% RSLogix 500 project LEGACY DRYER WITH LONOX AND SHUTDOWN DELAY.RSS, saved by version 11.00.00.00 %
PROJECT "ML1200"    % processor: MicroLogix 1200; MAIN_PROG %

PROGRAM FILES
  LAD 2 "MAIN_PROG"  15 rungs
  LAD 3 "DRYER CONT"  18 rungs
  LAD 4 "TEMPERATUR"  33 rungs
  LAD 5 "AIR PRES."  12 rungs
  LAD 6 "HUMIDITY"  14 rungs
  LAD 7 "RHL-TEMP"  2 rungs  % HEATING CONTROLS %
  LAD 8 "HEAT CONTR"  47 rungs
  LAD 9 "CLR FAULTS"  2 rungs
  LAD 10 "HOUR METER"  5 rungs
  LAD 11 "CONV CLEAN"  14 rungs

DATA FILES
  O0 OUTPUT  8 elements
  I1 INPUT  19 elements
  S2 STATUS  66 elements
  B3 BINARY  20 elements
  T4 TIMER  13 elements
  C5 COUNTER  1 elements
  R6 CONTROL  1 elements
  N7 INTEGER  77 elements
  F8 FLOAT  1 elements
  PD9 DRYER  3 elements

LADDER 2 "MAIN_PROG"
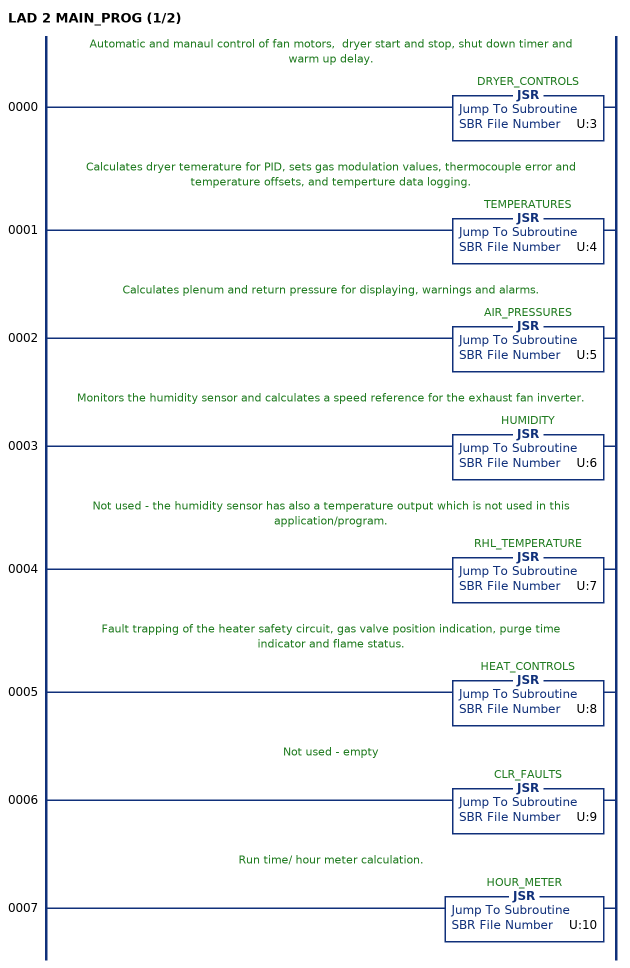
% Rung: 0 %
% Automatic and manaul control of fan motors,  dryer start and stop, shut down timer and warm up delay. %
SOR JSR U:3 EOR
%   U:3  DRYER_CONTROLS %
% Rung: 1 %
% Calculates dryer temerature for PID, sets gas modulation values, thermocouple error and temperature offsets, and temperture data logging. %
SOR JSR U:4 EOR
%   U:4  TEMPERATURES %
% Rung: 2 %
% Calculates plenum and return pressure for displaying, warnings and alarms. %
SOR JSR U:5 EOR
%   U:5  AIR_PRESSURES %
% Rung: 3 %
% Monitors the humidity sensor and calculates a speed reference for the exhaust fan inverter. %
SOR JSR U:6 EOR
%   U:6  HUMIDITY %
% Rung: 4 %
% Not used - the humidity sensor has also a temperature output which is not used in this application/program. %
SOR JSR U:7 EOR
%   U:7  RHL_TEMPERATURE %
% Rung: 5 %
% Fault trapping of the heater safety circuit, gas valve position indication, purge time indicator and flame status. %
SOR JSR U:8 EOR
%   U:8  HEAT_CONTROLS %
% Rung: 6 %
% Not used - empty %
SOR JSR U:9 EOR
%   U:9  CLR_FAULTS %
% Rung: 7 %
% Run time/ hour meter calculation. %
SOR JSR U:10 EOR
%   U:10  HOUR_METER %

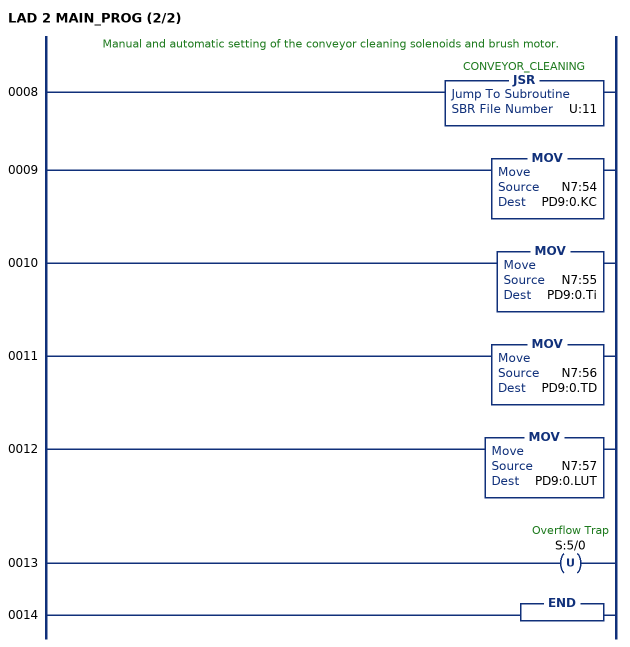
% Rung: 8 %
% Manual and automatic setting of the conveyor cleaning solenoids and brush motor. %
SOR JSR U:11 EOR
%   U:11  CONVEYOR_CLEANING %
% Rung: 9 %
SOR MOV N7:54 PD9:0.KC EOR
%   N7:54  KC %
% Rung: 10 %
SOR MOV N7:55 PD9:0.Ti EOR
%   N7:55  TI %
% Rung: 11 %
SOR MOV N7:56 PD9:0.TD EOR
%   N7:56  TD %
% Rung: 12 %
SOR MOV N7:57 PD9:0.LUT EOR
%   N7:57  LUT %
% Rung: 13 %
SOR OTU S:5/0 EOR
%   S:5/0  "Overflow Trap" %
% Rung: 14 %
SOR END EOR

LADDER 3 "DRYER CONT"
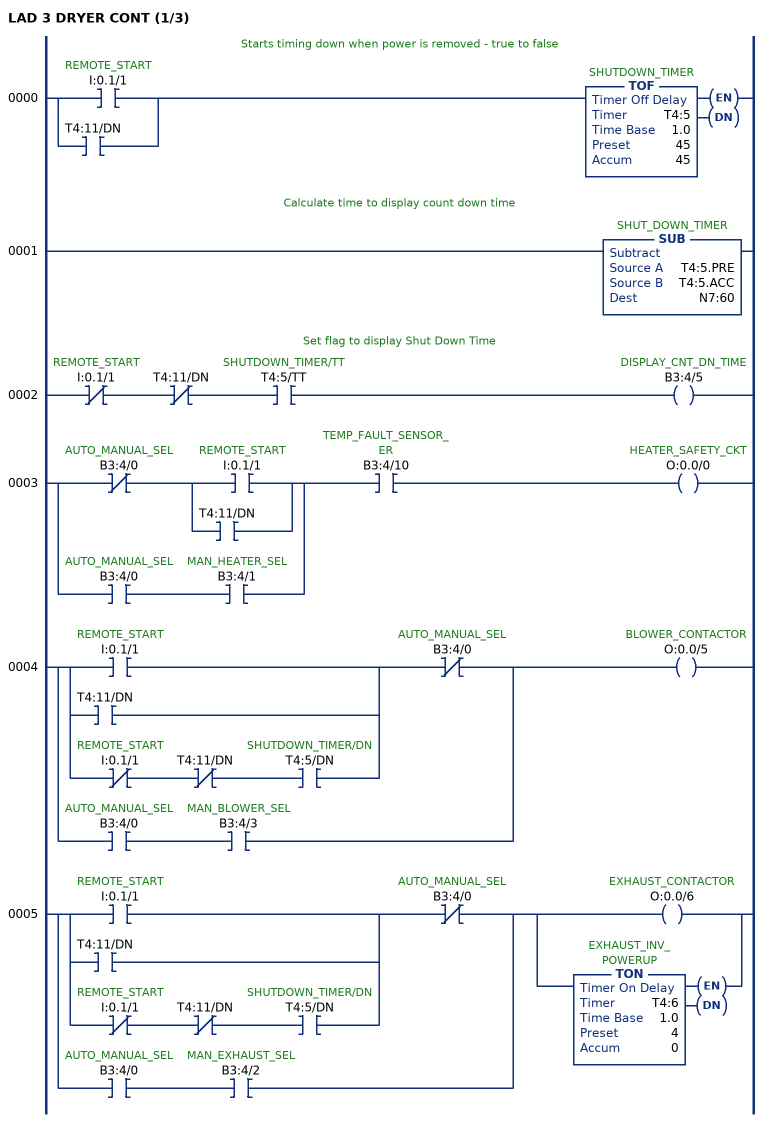
% Rung: 0 %
% Starts timing down when power is removed - true to false %
SOR BST XIC I:0.1/1 NXB XIC T4:11/DN BND TOF T4:5 1.0 45 45 EOR
%   I:0.1/1  REMOTE_START %
%   T4:5  SHUTDOWN_TIMER %
% Rung: 1 %
% Calculate time to display count down time %
SOR SUB T4:5.PRE T4:5.ACC N7:60 EOR
%   T4:5  SHUTDOWN_TIMER %
%   N7:60  SHUT_DOWN_TIMER %
% Rung: 2 %
% Set flag to display Shut Down Time %
SOR XIO I:0.1/1 XIO T4:11/DN XIC T4:5/TT OTE B3:4/5 EOR
%   I:0.1/1  REMOTE_START %
%   T4:5  SHUTDOWN_TIMER %
%   B3:4/5  DISPLAY_CNT_DN_TIME %
% Rung: 3 %
SOR BST XIO B3:4/0 BST XIC I:0.1/1 NXB XIC T4:11/DN BND NXB XIC B3:4/0 XIC B3:4/1 BND XIC B3:4/10 OTE O:0.0/0 EOR
%   B3:4/0  AUTO_MANUAL_SEL %
%   I:0.1/1  REMOTE_START %
%   B3:4/1  MAN_HEATER_SEL %
%   B3:4/10  TEMP_FAULT_SENSOR_ER %
%   O:0.0/0  HEATER_SAFETY_CKT %
% Rung: 4 %
SOR BST BST BST XIC I:0.1/1 NXB XIC T4:11/DN BND NXB XIO I:0.1/1 XIO T4:11/DN XIC T4:5/DN BND XIO B3:4/0 NXB XIC B3:4/0 XIC B3:4/3 BND OTE O:0.0/5 EOR
%   I:0.1/1  REMOTE_START %
%   T4:5  SHUTDOWN_TIMER %
%   B3:4/0  AUTO_MANUAL_SEL %
%   B3:4/3  MAN_BLOWER_SEL %
%   O:0.0/5  BLOWER_CONTACTOR %
% Rung: 5 %
SOR BST BST BST XIC I:0.1/1 NXB XIC T4:11/DN BND NXB XIO I:0.1/1 XIO T4:11/DN XIC T4:5/DN BND XIO B3:4/0 NXB XIC B3:4/0 XIC B3:4/2 BND BST OTE O:0.0/6 NXB TON T4:6 1.0 4 0 BND EOR
%   I:0.1/1  REMOTE_START %
%   T4:5  SHUTDOWN_TIMER %
%   B3:4/0  AUTO_MANUAL_SEL %
%   B3:4/2  MAN_EXHAUST_SEL %
%   O:0.0/6  EXHAUST_CONTACTOR %
%   T4:6  EXHAUST_INV_POWERUP %

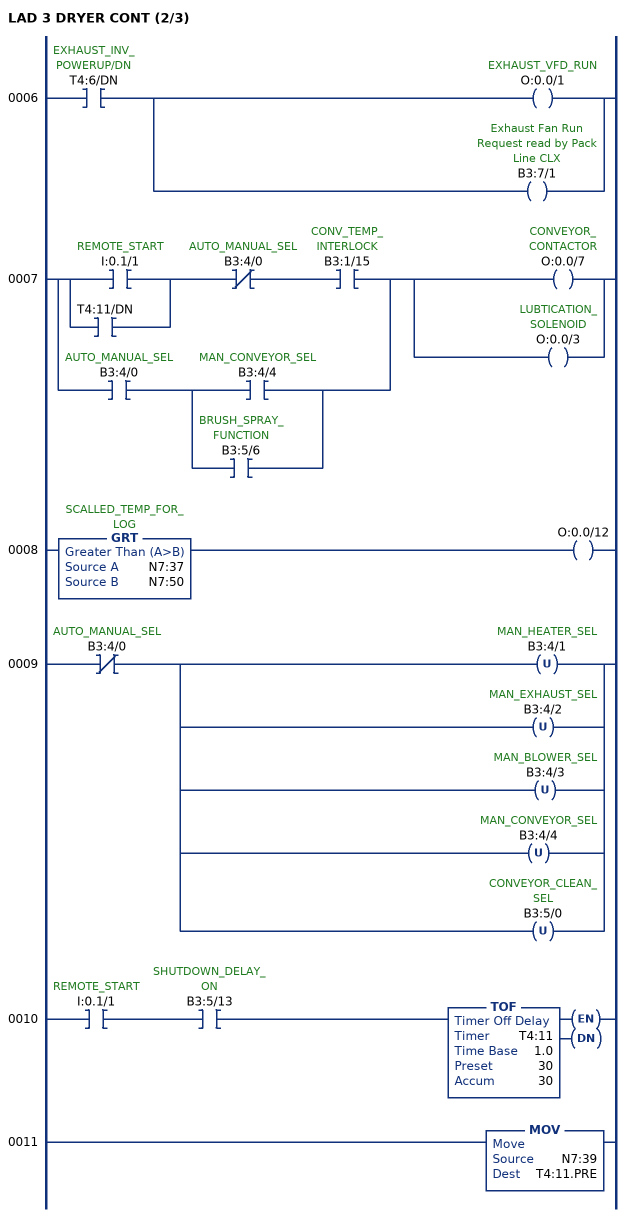
% Rung: 6 %
SOR XIC T4:6/DN BST OTE O:0.0/1 NXB OTE B3:7/1 BND EOR
%   T4:6  EXHAUST_INV_POWERUP %
%   O:0.0/1  EXHAUST_VFD_RUN %
%   B3:7/1  "Exhaust Fan Run Request read by Pack Line CLX" %
% Rung: 7 %
SOR BST BST XIC I:0.1/1 NXB XIC T4:11/DN BND XIO B3:4/0 XIC B3:1/15 NXB XIC B3:4/0 BST XIC B3:4/4 NXB XIC B3:5/6 BND BND BST OTE O:0.0/7 NXB OTE O:0.0/3 BND EOR
%   I:0.1/1  REMOTE_START %
%   B3:4/0  AUTO_MANUAL_SEL %
%   B3:1/15  CONV_TEMP_INTERLOCK %
%   B3:4/4  MAN_CONVEYOR_SEL %
%   B3:5/6  BRUSH_SPRAY_FUNCTION %
%   O:0.0/7  CONVEYOR_CONTACTOR %
%   O:0.0/3  LUBTICATION_SOLENOID %
% Rung: 8 %
SOR GRT N7:37 N7:50 OTE O:0.0/12 EOR
%   N7:37  SCALLED_TEMP_FOR_LOG %
% Rung: 9 %
SOR XIO B3:4/0 BST OTU B3:4/1 NXB BST OTU B3:4/2 NXB BST OTU B3:4/3 NXB BST OTU B3:4/4 NXB OTU B3:5/0 BND BND BND BND EOR
%   B3:4/0  AUTO_MANUAL_SEL %
%   B3:4/1  MAN_HEATER_SEL %
%   B3:4/2  MAN_EXHAUST_SEL %
%   B3:4/3  MAN_BLOWER_SEL %
%   B3:4/4  MAN_CONVEYOR_SEL %
%   B3:5/0  CONVEYOR_CLEAN_SEL %
% Rung: 10 %
SOR XIC I:0.1/1 XIC B3:5/13 TOF T4:11 1.0 30 30 EOR
%   I:0.1/1  REMOTE_START %
%   B3:5/13  SHUTDOWN_DELAY_ON %
% Rung: 11 %
SOR MOV N7:39 T4:11.PRE EOR

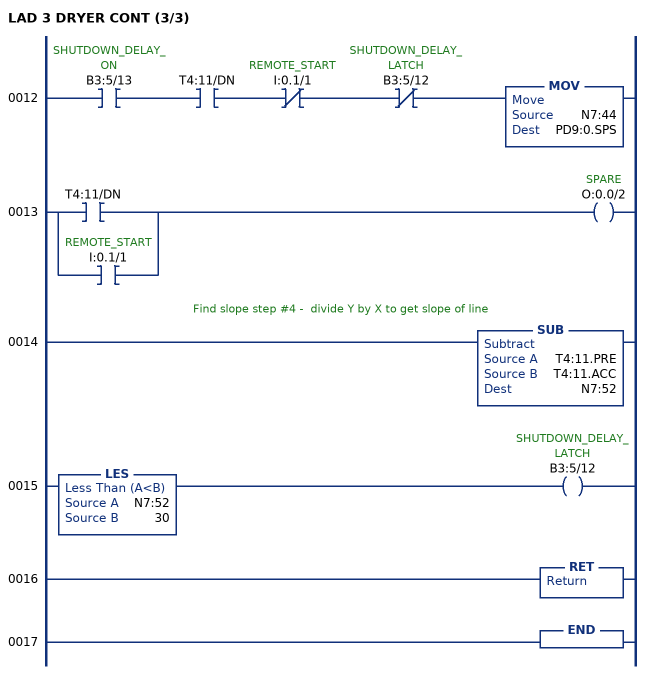
% Rung: 12 %
SOR XIC B3:5/13 XIC T4:11/DN XIO I:0.1/1 XIO B3:5/12 MOV N7:44 PD9:0.SPS EOR
%   B3:5/13  SHUTDOWN_DELAY_ON %
%   I:0.1/1  REMOTE_START %
%   B3:5/12  SHUTDOWN_DELAY_LATCH %
%   N7:44  TEMP_ON_SHUTDOWN_DLY %
% Rung: 13 %
SOR BST XIC T4:11/DN NXB XIC I:0.1/1 BND OTE O:0.0/2 EOR
%   I:0.1/1  REMOTE_START %
%   O:0.0/2  SPARE %
% Rung: 14 %
% Find slope step #4 -  divide Y by X to get slope of line %
SOR SUB T4:11.PRE T4:11.ACC N7:52 EOR
% Rung: 15 %
SOR LES N7:52 30 OTE B3:5/12 EOR
%   B3:5/12  SHUTDOWN_DELAY_LATCH %
% Rung: 16 %
SOR RET EOR
% Rung: 17 %
SOR END EOR

LADDER 4 "TEMPERATUR"
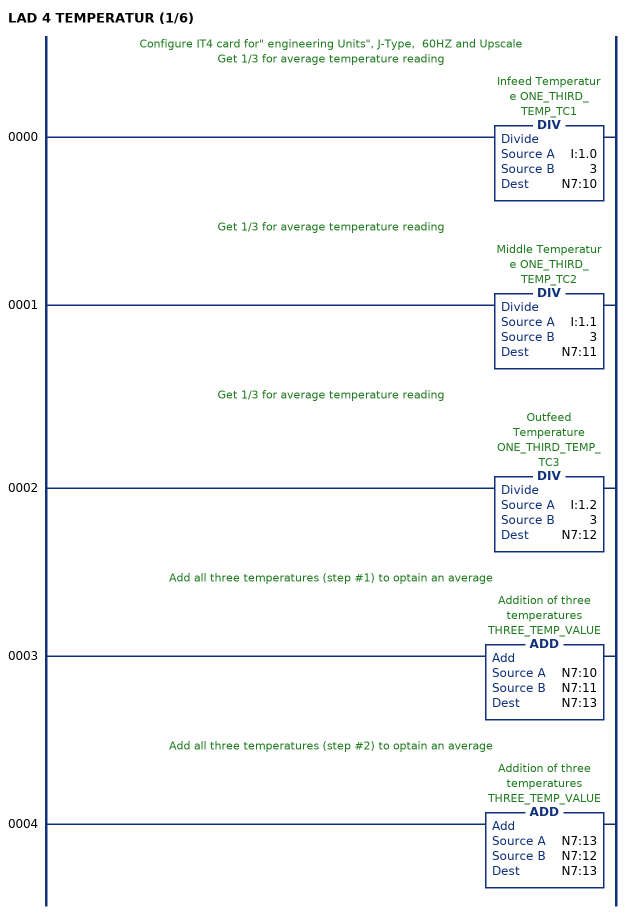
% Rung: 0 %
% Configure IT4 card for" engineering Units", J-Type,  60HZ and Upscale
% Get 1/3 for average temperature reading %
SOR DIV I:1.0 3 N7:10 EOR
%   I:1.0  INFEED_TEMP %
%   N7:10  ONE_THIRD_TEMP_TC1  "Infeed Temperature" %
% Rung: 1 %
% Get 1/3 for average temperature reading %
SOR DIV I:1.1 3 N7:11 EOR
%   I:1.1  MIDDLE_TEMP %
%   N7:11  ONE_THIRD_TEMP_TC2  "Middle Temperature" %
% Rung: 2 %
% Get 1/3 for average temperature reading %
SOR DIV I:1.2 3 N7:12 EOR
%   I:1.2  OUTFEED_TEMP %
%   N7:12  ONE_THIRD_TEMP_TC3  "Outfeed Temperature" %
% Rung: 3 %
% Add all three temperatures (step #1) to optain an average %
SOR ADD N7:10 N7:11 N7:13 EOR
%   N7:10  ONE_THIRD_TEMP_TC1  "Infeed Temperature" %
%   N7:11  ONE_THIRD_TEMP_TC2  "Middle Temperature" %
%   N7:13  THREE_TEMP_VALUE  "Addition of three temperatures" %
% Rung: 4 %
% Add all three temperatures (step #2) to optain an average %
SOR ADD N7:13 N7:12 N7:13 EOR
%   N7:13  THREE_TEMP_VALUE  "Addition of three temperatures" %
%   N7:12  ONE_THIRD_TEMP_TC3  "Outfeed Temperature" %

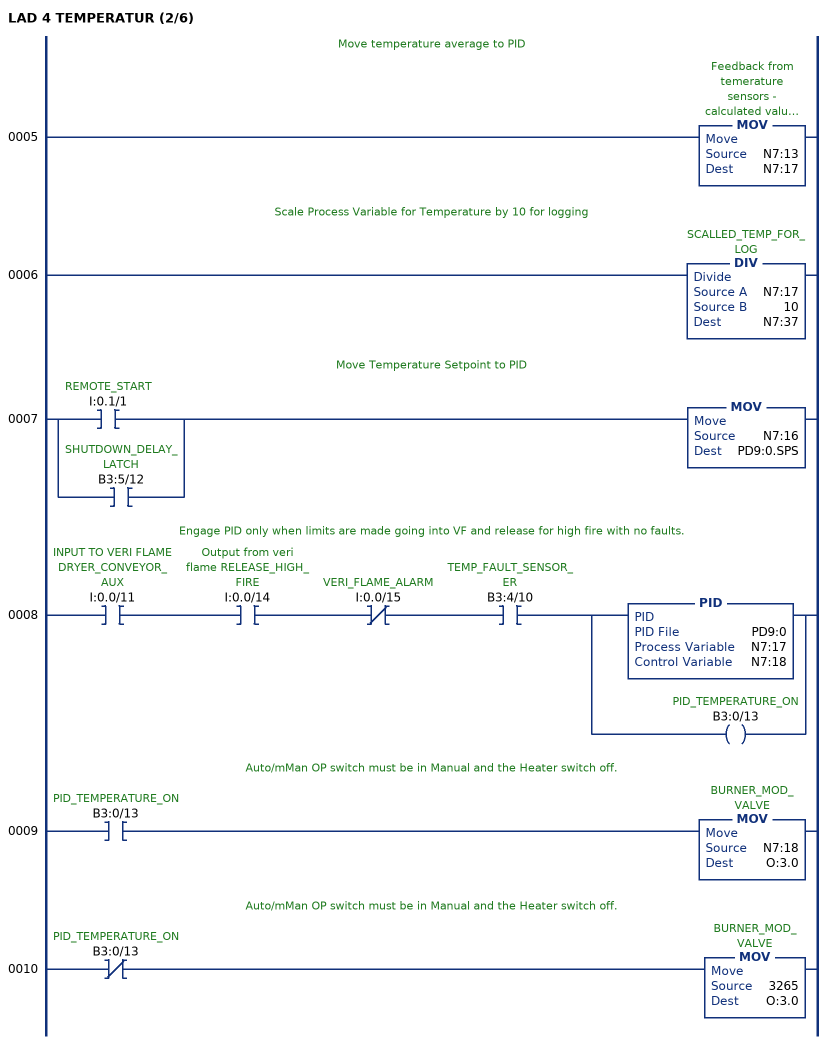
% Rung: 5 %
% Move temperature average to PID %
SOR MOV N7:13 N7:17 EOR
%   N7:13  THREE_TEMP_VALUE  "Addition of three temperatures" %
%   N7:17  PV_TEMP_PROCESS_VAR  "Feedback from temerature sensors - calculated value" %
% Rung: 6 %
% Scale Process Variable for Temperature by 10 for logging %
SOR DIV N7:17 10 N7:37 EOR
%   N7:17  PV_TEMP_PROCESS_VAR  "Feedback from temerature sensors - calculated value" %
%   N7:37  SCALLED_TEMP_FOR_LOG %
% Rung: 7 %
% Move Temperature Setpoint to PID %
SOR BST XIC I:0.1/1 NXB XIC B3:5/12 BND MOV N7:16 PD9:0.SPS EOR
%   I:0.1/1  REMOTE_START %
%   B3:5/12  SHUTDOWN_DELAY_LATCH %
%   N7:16  SPS_TEMP_SETPOINT  "Display Input Value - desired Temperature" %
% Rung: 8 %
% Engage PID only when limits are made going into VF and release for high fire with no faults. %
SOR XIC I:0.0/11 XIC I:0.0/14 XIO I:0.0/15 XIC B3:4/10 BST PID PD9:0 N7:17 N7:18 NXB OTE B3:0/13 BND EOR
%   I:0.0/11  DRYER_CONVEYOR_AUX  "INPUT TO VERI FLAME" %
%   I:0.0/14  RELEASE_HIGH_FIRE  "Output from veri flame" %
%   I:0.0/15  VERI_FLAME_ALARM %
%   B3:4/10  TEMP_FAULT_SENSOR_ER %
%   N7:17  PV_TEMP_PROCESS_VAR  "Feedback from temerature sensors - calculated value" %
%   N7:18  CV_TEMP_CONTROL_VAR  "Output value to output for output card" %
%   B3:0/13  PID_TEMPERATURE_ON %
% Rung: 9 %
% Auto/mMan OP switch must be in Manual and the Heater switch off. %
SOR XIC B3:0/13 MOV N7:18 O:3.0 EOR
%   B3:0/13  PID_TEMPERATURE_ON %
%   N7:18  CV_TEMP_CONTROL_VAR  "Output value to output for output card" %
%   O:3.0  BURNER_MOD_VALVE %
% Rung: 10 %
% Auto/mMan OP switch must be in Manual and the Heater switch off. %
SOR XIO B3:0/13 MOV 3265 O:3.0 EOR
%   B3:0/13  PID_TEMPERATURE_ON %
%   O:3.0  BURNER_MOD_VALVE %

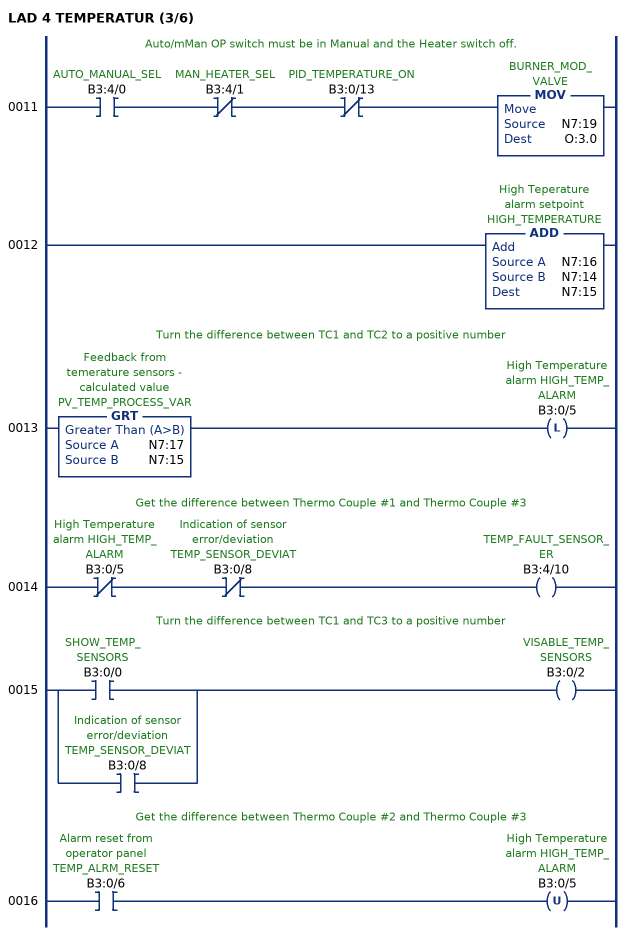
% Rung: 11 %
% Auto/mMan OP switch must be in Manual and the Heater switch off. %
SOR XIC B3:4/0 XIO B3:4/1 XIO B3:0/13 MOV N7:19 O:3.0 EOR
%   B3:4/0  AUTO_MANUAL_SEL %
%   B3:4/1  MAN_HEATER_SEL %
%   B3:0/13  PID_TEMPERATURE_ON %
%   N7:19  MANUAL_GAS_VALVE_POS  "To test burner butterfly in Manual" %
%   O:3.0  BURNER_MOD_VALVE %
% Rung: 12 %
SOR ADD N7:16 N7:14 N7:15 EOR
%   N7:16  SPS_TEMP_SETPOINT  "Display Input Value - desired Temperature" %
%   N7:14  HIGH_TEMP_OFFSET  "Value added to Temp Setpoint to set high temerature" %
%   N7:15  HIGH_TEMPERATURE  "High Teperature alarm setpoint" %
% Rung: 13 %
% Turn the difference between TC1 and TC2 to a positive number %
SOR GRT N7:17 N7:15 OTL B3:0/5 EOR
%   N7:17  PV_TEMP_PROCESS_VAR  "Feedback from temerature sensors - calculated value" %
%   N7:15  HIGH_TEMPERATURE  "High Teperature alarm setpoint" %
%   B3:0/5  HIGH_TEMP_ALARM  "High Temperature alarm" %
% Rung: 14 %
% Get the difference between Thermo Couple #1 and Thermo Couple #3 %
SOR XIO B3:0/5 XIO B3:0/8 OTE B3:4/10 EOR
%   B3:0/5  HIGH_TEMP_ALARM  "High Temperature alarm" %
%   B3:0/8  TEMP_SENSOR_DEVIAT  "Indication of sensor error/deviation" %
%   B3:4/10  TEMP_FAULT_SENSOR_ER %
% Rung: 15 %
% Turn the difference between TC1 and TC3 to a positive number %
SOR BST XIC B3:0/0 NXB XIC B3:0/8 BND OTE B3:0/2 EOR
%   B3:0/0  SHOW_TEMP_SENSORS %
%   B3:0/8  TEMP_SENSOR_DEVIAT  "Indication of sensor error/deviation" %
%   B3:0/2  VISABLE_TEMP_SENSORS %
% Rung: 16 %
% Get the difference between Thermo Couple #2 and Thermo Couple #3 %
SOR XIC B3:0/6 OTU B3:0/5 EOR
%   B3:0/6  TEMP_ALRM_RESET  "Alarm reset from operator panel" %
%   B3:0/5  HIGH_TEMP_ALARM  "High Temperature alarm" %

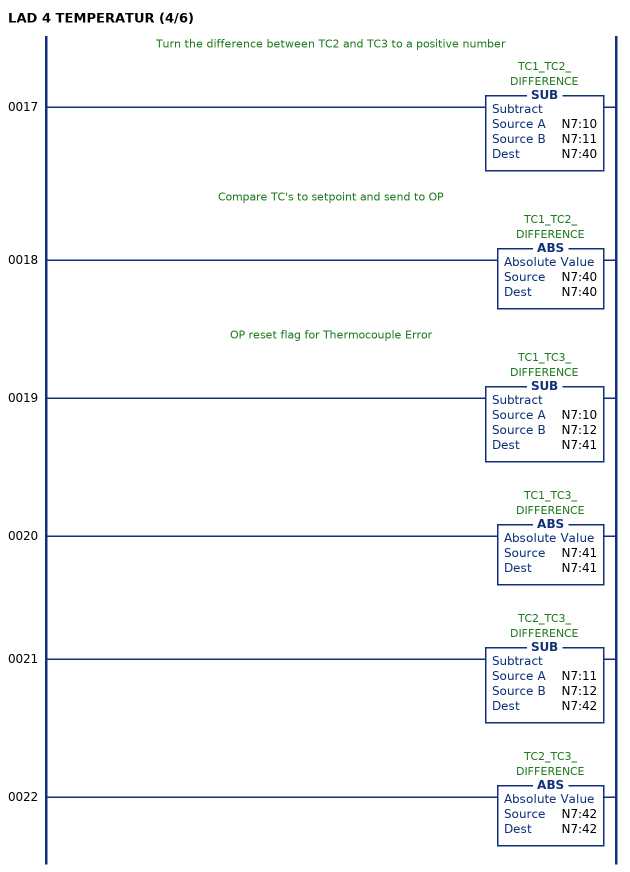
% Rung: 17 %
% Turn the difference between TC2 and TC3 to a positive number %
SOR SUB N7:10 N7:11 N7:40 EOR
%   N7:10  ONE_THIRD_TEMP_TC1  "Infeed Temperature" %
%   N7:11  ONE_THIRD_TEMP_TC2  "Middle Temperature" %
%   N7:40  TC1_TC2_DIFFERENCE %
% Rung: 18 %
% Compare TC's to setpoint and send to OP %
SOR ABS N7:40 N7:40 EOR
%   N7:40  TC1_TC2_DIFFERENCE %
% Rung: 19 %
% OP reset flag for Thermocouple Error %
SOR SUB N7:10 N7:12 N7:41 EOR
%   N7:10  ONE_THIRD_TEMP_TC1  "Infeed Temperature" %
%   N7:12  ONE_THIRD_TEMP_TC3  "Outfeed Temperature" %
%   N7:41  TC1_TC3_DIFFERENCE %
% Rung: 20 %
SOR ABS N7:41 N7:41 EOR
%   N7:41  TC1_TC3_DIFFERENCE %
% Rung: 21 %
SOR SUB N7:11 N7:12 N7:42 EOR
%   N7:11  ONE_THIRD_TEMP_TC2  "Middle Temperature" %
%   N7:12  ONE_THIRD_TEMP_TC3  "Outfeed Temperature" %
%   N7:42  TC2_TC3_DIFFERENCE %
% Rung: 22 %
SOR ABS N7:42 N7:42 EOR
%   N7:42  TC2_TC3_DIFFERENCE %

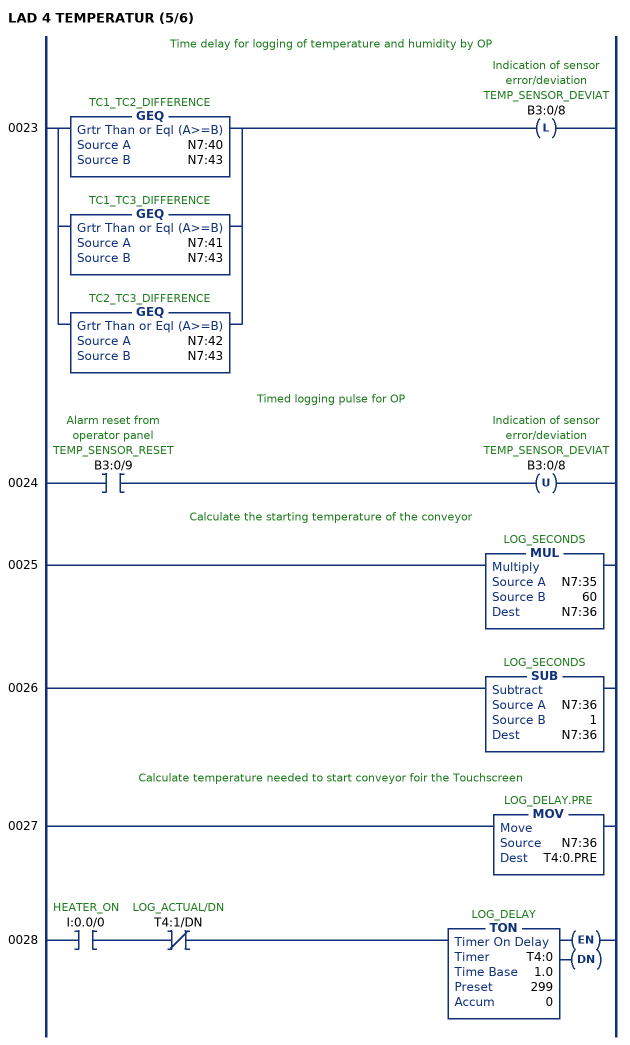
% Rung: 23 %
% Time delay for logging of temperature and humidity by OP %
SOR BST GEQ N7:40 N7:43 NXB BST GEQ N7:41 N7:43 NXB GEQ N7:42 N7:43 BND BND OTL B3:0/8 EOR
%   N7:40  TC1_TC2_DIFFERENCE %
%   N7:43  MAX_TEMP_SENSOR_DEV %
%   N7:41  TC1_TC3_DIFFERENCE %
%   N7:42  TC2_TC3_DIFFERENCE %
%   B3:0/8  TEMP_SENSOR_DEVIAT  "Indication of sensor error/deviation" %
% Rung: 24 %
% Timed logging pulse for OP %
SOR XIC B3:0/9 OTU B3:0/8 EOR
%   B3:0/9  TEMP_SENSOR_RESET  "Alarm reset from operator panel" %
%   B3:0/8  TEMP_SENSOR_DEVIAT  "Indication of sensor error/deviation" %
% Rung: 25 %
% Calculate the starting temperature of the conveyor %
SOR MUL N7:35 60 N7:36 EOR
%   N7:35  LOG_MINUTES %
%   N7:36  LOG_SECONDS %
% Rung: 26 %
SOR SUB N7:36 1 N7:36 EOR
%   N7:36  LOG_SECONDS %
% Rung: 27 %
% Calculate temperature needed to start conveyor foir the Touchscreen %
SOR MOV N7:36 T4:0.PRE EOR
%   N7:36  LOG_SECONDS %
%   T4:0  LOG_DELAY %
% Rung: 28 %
SOR XIC I:0.0/0 XIO T4:1/DN TON T4:0 1.0 299 0 EOR
%   I:0.0/0  HEATER_ON %
%   T4:1  LOG_ACTUAL %
%   T4:0  LOG_DELAY %

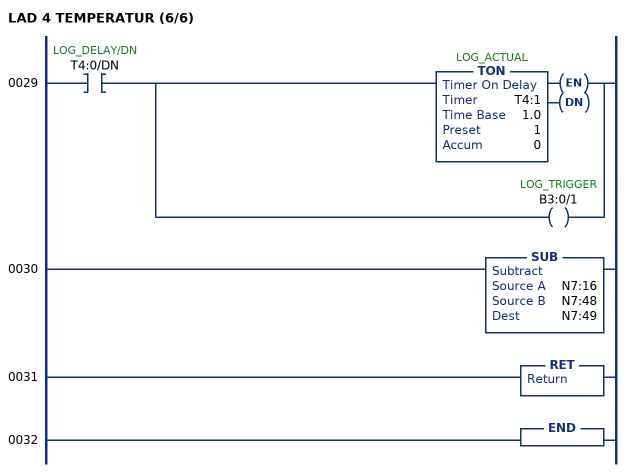
% Rung: 29 %
SOR XIC T4:0/DN BST TON T4:1 1.0 1 0 NXB OTE B3:0/1 BND EOR
%   T4:0  LOG_DELAY %
%   T4:1  LOG_ACTUAL %
%   B3:0/1  LOG_TRIGGER %
% Rung: 30 %
SOR SUB N7:16 N7:48 N7:49 EOR
%   N7:16  SPS_TEMP_SETPOINT  "Display Input Value - desired Temperature" %
% Rung: 31 %
SOR RET EOR
% Rung: 32 %
SOR END EOR

LADDER 5 "AIR PRES."
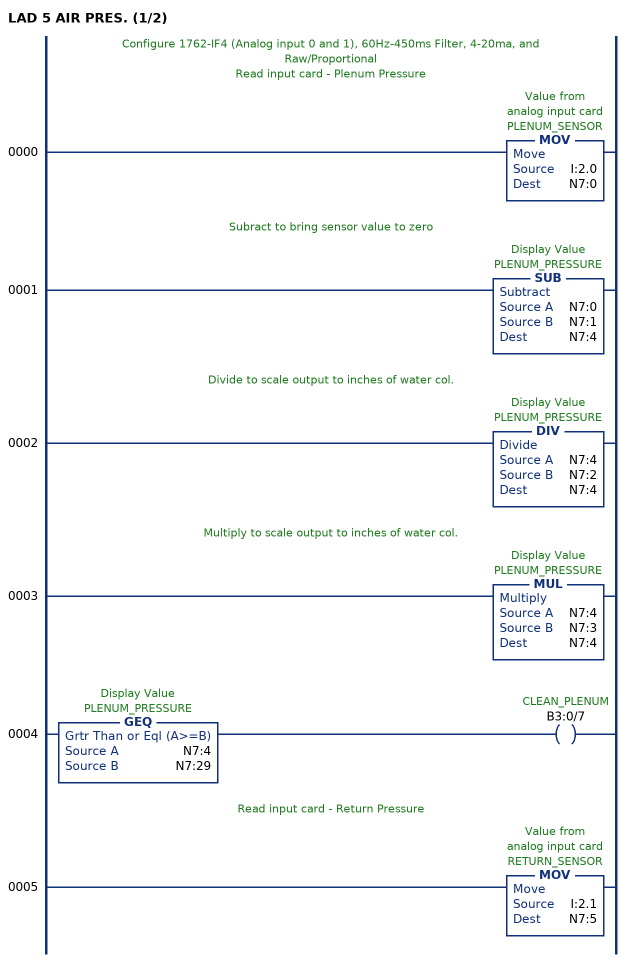
% Rung: 0 %
% Configure 1762-IF4 (Analog input 0 and 1), 60Hz-450ms Filter, 4-20ma, and Raw/Proportional
% Read input card - Plenum Pressure %
SOR MOV I:2.0 N7:0 EOR
%   N7:0  PLENUM_SENSOR  "Value from analog input card" %
% Rung: 1 %
% Subract to bring sensor value to zero %
SOR SUB N7:0 N7:1 N7:4 EOR
%   N7:0  PLENUM_SENSOR  "Value from analog input card" %
%   N7:1  PLENUM_ZERO  "The amount needed to return a zero value with no pressure" %
%   N7:4  PLENUM_PRESSURE  "Display Value" %
% Rung: 2 %
% Divide to scale output to inches of water col. %
SOR DIV N7:4 N7:2 N7:4 EOR
%   N7:4  PLENUM_PRESSURE  "Display Value" %
%   N7:2  PLENUM_SCALING_DIV  "Value needed to adjust output to meter range" %
% Rung: 3 %
% Multiply to scale output to inches of water col. %
SOR MUL N7:4 N7:3 N7:4 EOR
%   N7:4  PLENUM_PRESSURE  "Display Value" %
%   N7:3  PLENUM_SCALING_MUL  "Value needed to adjust output to meter range" %
% Rung: 4 %
SOR GEQ N7:4 N7:29 OTE B3:0/7 EOR
%   N7:4  PLENUM_PRESSURE  "Display Value" %
%   N7:29  PLENUM_ALARM  "signal Operator Panel that cleaning is required" %
%   B3:0/7  CLEAN_PLENUM %
% Rung: 5 %
% Read input card - Return Pressure %
SOR MOV I:2.1 N7:5 EOR
%   N7:5  RETURN_SENSOR  "Value from analog input card" %

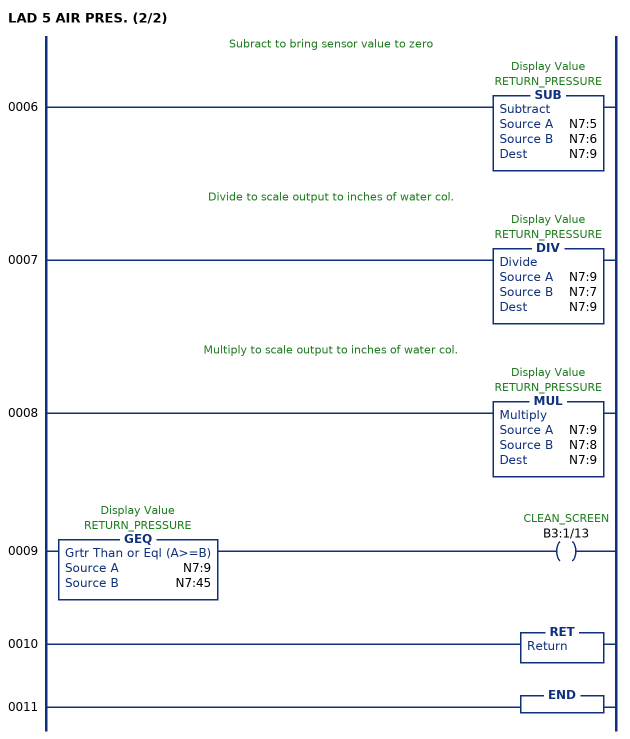
% Rung: 6 %
% Subract to bring sensor value to zero %
SOR SUB N7:5 N7:6 N7:9 EOR
%   N7:5  RETURN_SENSOR  "Value from analog input card" %
%   N7:6  RETURN_ZERO  "The amount needed to return a zero value with no pressure" %
%   N7:9  RETURN_PRESSURE  "Display Value" %
% Rung: 7 %
% Divide to scale output to inches of water col. %
SOR DIV N7:9 N7:7 N7:9 EOR
%   N7:9  RETURN_PRESSURE  "Display Value" %
%   N7:7  RETURN_SCALING  "Value needed to adjust output to meter range" %
% Rung: 8 %
% Multiply to scale output to inches of water col. %
SOR MUL N7:9 N7:8 N7:9 EOR
%   N7:9  RETURN_PRESSURE  "Display Value" %
%   N7:8  RETURN_SCALING_MUL  "Value needed to adjust output to meter range" %
% Rung: 9 %
SOR GEQ N7:9 N7:45 OTE B3:1/13 EOR
%   N7:9  RETURN_PRESSURE  "Display Value" %
%   N7:45  CLEAN_SCREEN_ALARM %
%   B3:1/13  CLEAN_SCREEN %
% Rung: 10 %
SOR RET EOR
% Rung: 11 %
SOR END EOR

LADDER 6 "HUMIDITY"
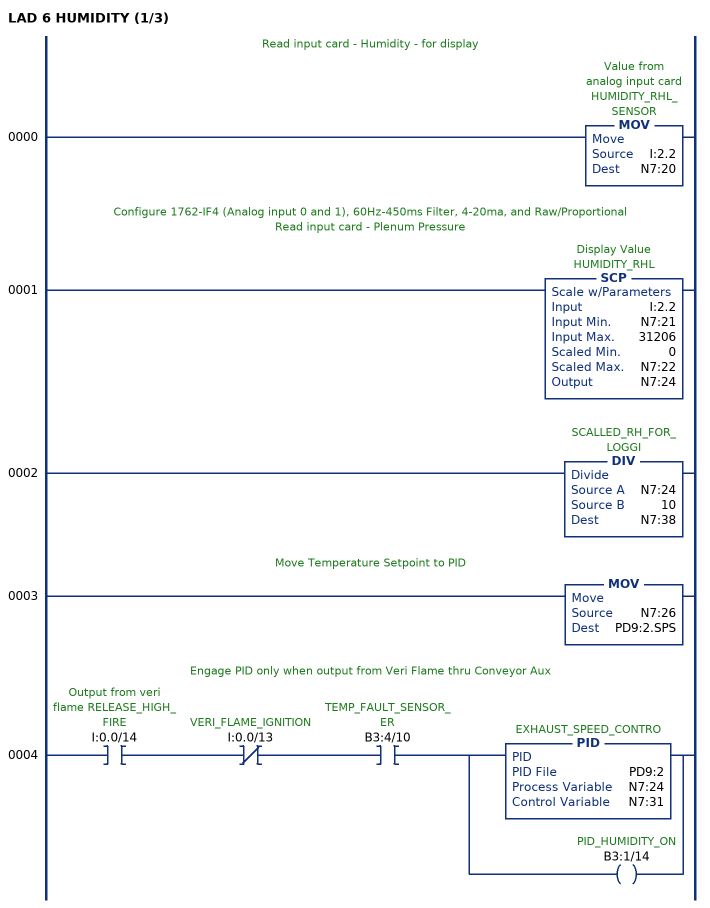
% Rung: 0 %
% Read input card - Humidity - for display %
SOR MOV I:2.2 N7:20 EOR
%   N7:20  HUMIDITY_RHL_SENSOR  "Value from analog input card" %
% Rung: 1 %
% Configure 1762-IF4 (Analog input 0 and 1), 60Hz-450ms Filter, 4-20ma, and Raw/Proportional
% Read input card - Plenum Pressure %
SOR SCP I:2.2 N7:21 31206 0 N7:22 N7:24 EOR
%   N7:21  HUMIDITY_ZERO  "The amount needed to return a zero value with no humitity" %
%   N7:22  HUMIDITY_SCALING_MAX  "Max range of sensor" %
%   N7:24  HUMIDITY_RHL  "Display Value" %
% Rung: 2 %
SOR DIV N7:24 10 N7:38 EOR
%   N7:24  HUMIDITY_RHL  "Display Value" %
%   N7:38  SCALLED_RH_FOR_LOGGI %
% Rung: 3 %
% Move Temperature Setpoint to PID %
SOR MOV N7:26 PD9:2.SPS EOR
%   N7:26  HUMITITY_MAX_SETPOIN %
% Rung: 4 %
% Engage PID only when output from Veri Flame thru Conveyor Aux %
SOR XIC I:0.0/14 XIO I:0.0/13 XIC B3:4/10 BST PID PD9:2 N7:24 N7:31 NXB OTE B3:1/14 BND EOR
%   I:0.0/14  RELEASE_HIGH_FIRE  "Output from veri flame" %
%   I:0.0/13  VERI_FLAME_IGNITION %
%   B3:4/10  TEMP_FAULT_SENSOR_ER %
%   PD9:2  EXHAUST_SPEED_CONTRO %
%   N7:24  HUMIDITY_RHL  "Display Value" %
%   N7:31  CV_RH_CONTROL_VAR  "Output value to output for output card" %
%   B3:1/14  PID_HUMIDITY_ON %

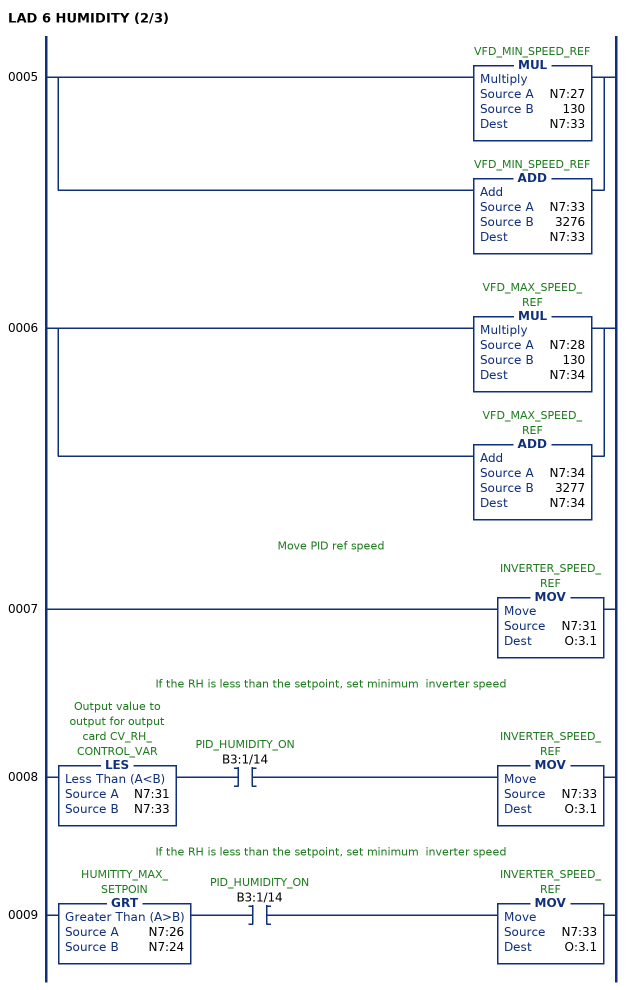
% Rung: 5 %
SOR BST MUL N7:27 130 N7:33 NXB ADD N7:33 3276 N7:33 BND EOR
%   N7:27  EXHAUST_MIN_SPEED %
%   N7:33  VFD_MIN_SPEED_REF %
% Rung: 6 %
SOR BST MUL N7:28 130 N7:34 NXB ADD N7:34 3277 N7:34 BND EOR
%   N7:28  EXHAUST_MAX_SPEED %
%   N7:34  VFD_MAX_SPEED_REF %
% Rung: 7 %
% Move PID ref speed %
SOR MOV N7:31 O:3.1 EOR
%   N7:31  CV_RH_CONTROL_VAR  "Output value to output for output card" %
%   O:3.1  INVERTER_SPEED_REF %
% Rung: 8 %
% If the RH is less than the setpoint, set minimum  inverter speed %
SOR LES N7:31 N7:33 XIC B3:1/14 MOV N7:33 O:3.1 EOR
%   N7:31  CV_RH_CONTROL_VAR  "Output value to output for output card" %
%   N7:33  VFD_MIN_SPEED_REF %
%   B3:1/14  PID_HUMIDITY_ON %
%   O:3.1  INVERTER_SPEED_REF %
% Rung: 9 %
% If the RH is less than the setpoint, set minimum  inverter speed %
SOR GRT N7:26 N7:24 XIC B3:1/14 MOV N7:33 O:3.1 EOR
%   N7:26  HUMITITY_MAX_SETPOIN %
%   N7:24  HUMIDITY_RHL  "Display Value" %
%   B3:1/14  PID_HUMIDITY_ON %
%   N7:33  VFD_MIN_SPEED_REF %
%   O:3.1  INVERTER_SPEED_REF %

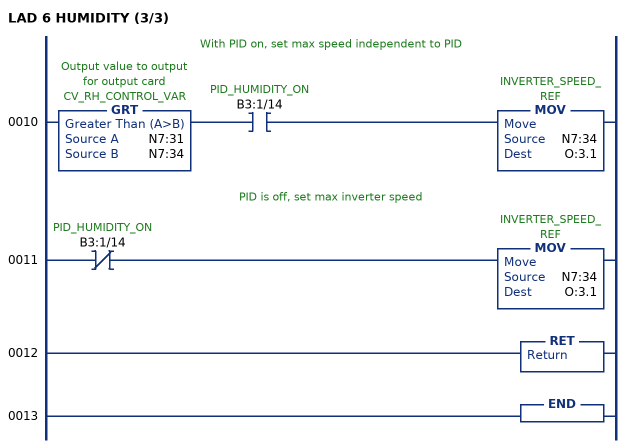
% Rung: 10 %
% With PID on, set max speed independent to PID %
SOR GRT N7:31 N7:34 XIC B3:1/14 MOV N7:34 O:3.1 EOR
%   N7:31  CV_RH_CONTROL_VAR  "Output value to output for output card" %
%   N7:34  VFD_MAX_SPEED_REF %
%   B3:1/14  PID_HUMIDITY_ON %
%   O:3.1  INVERTER_SPEED_REF %
% Rung: 11 %
% PID is off, set max inverter speed %
SOR XIO B3:1/14 MOV N7:34 O:3.1 EOR
%   B3:1/14  PID_HUMIDITY_ON %
%   N7:34  VFD_MAX_SPEED_REF %
%   O:3.1  INVERTER_SPEED_REF %
% Rung: 12 %
SOR RET EOR
% Rung: 13 %
SOR END EOR

LADDER 7 "RHL-TEMP"    % HEATING CONTROLS %
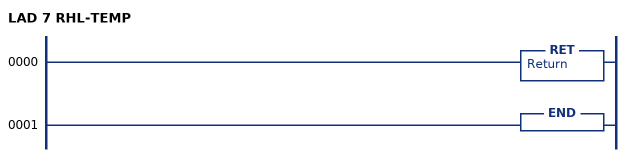
% Rung: 0 %
SOR RET EOR
% Rung: 1 %
SOR END EOR

LADDER 8 "HEAT CONTR"
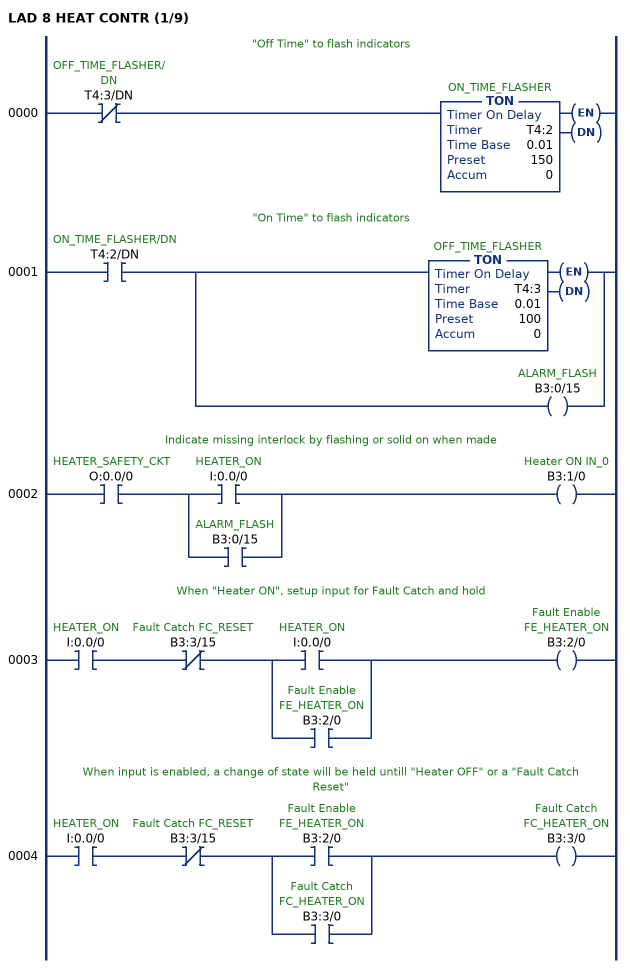
% Rung: 0 %
% "Off Time" to flash indicators %
SOR XIO T4:3/DN TON T4:2 0.01 150 0 EOR
%   T4:3  OFF_TIME_FLASHER %
%   T4:2  ON_TIME_FLASHER %
% Rung: 1 %
% "On Time" to flash indicators %
SOR XIC T4:2/DN BST TON T4:3 0.01 100 0 NXB OTE B3:0/15 BND EOR
%   T4:2  ON_TIME_FLASHER %
%   T4:3  OFF_TIME_FLASHER %
%   B3:0/15  ALARM_FLASH %
% Rung: 2 %
% Indicate missing interlock by flashing or solid on when made %
SOR XIC O:0.0/0 BST XIC I:0.0/0 NXB XIC B3:0/15 BND OTE B3:1/0 EOR
%   O:0.0/0  HEATER_SAFETY_CKT %
%   I:0.0/0  HEATER_ON %
%   B3:0/15  ALARM_FLASH %
%   B3:1/0  IN_0  "Heater ON" %
% Rung: 3 %
% When "Heater ON", setup input for Fault Catch and hold %
SOR XIC I:0.0/0 XIO B3:3/15 BST XIC I:0.0/0 NXB XIC B3:2/0 BND OTE B3:2/0 EOR
%   I:0.0/0  HEATER_ON %
%   B3:3/15  FC_RESET  "Fault Catch" %
%   B3:2/0  FE_HEATER_ON  "Fault Enable" %
% Rung: 4 %
% When input is enabled, a change of state will be held untill "Heater OFF" or a "Fault Catch Reset" %
SOR XIC I:0.0/0 XIO B3:3/15 BST XIC B3:2/0 NXB XIC B3:3/0 BND OTE B3:3/0 EOR
%   I:0.0/0  HEATER_ON %
%   B3:3/15  FC_RESET  "Fault Catch" %
%   B3:2/0  FE_HEATER_ON  "Fault Enable" %
%   B3:3/0  FC_HEATER_ON  "Fault Catch" %

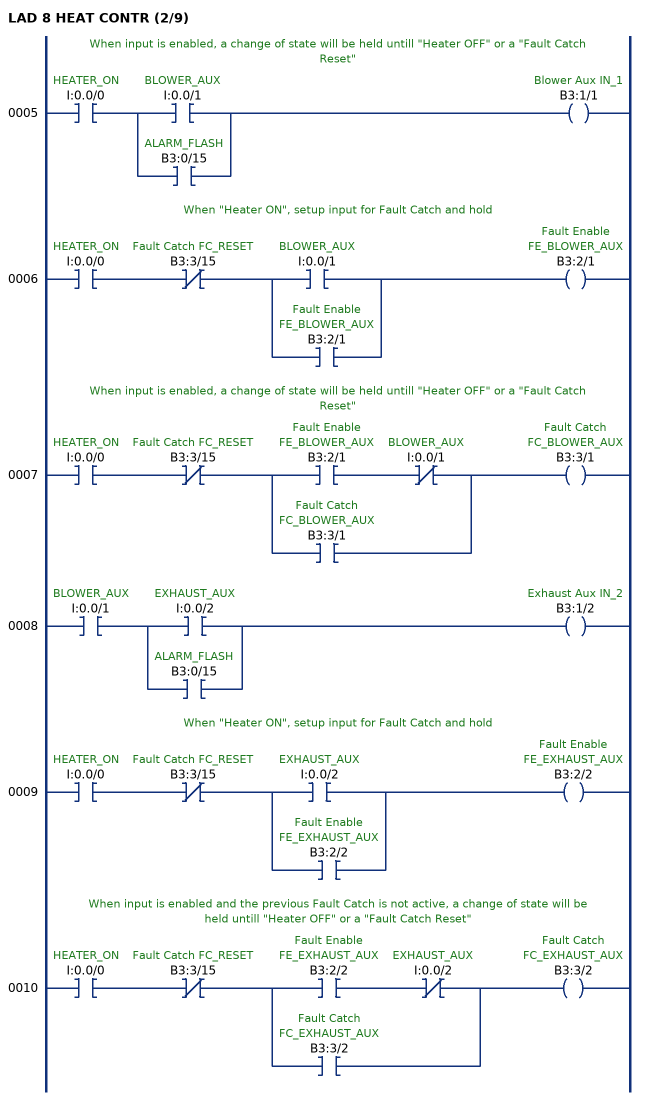
% Rung: 5 %
% When input is enabled, a change of state will be held untill "Heater OFF" or a "Fault Catch Reset" %
SOR XIC I:0.0/0 BST XIC I:0.0/1 NXB XIC B3:0/15 BND OTE B3:1/1 EOR
%   I:0.0/0  HEATER_ON %
%   I:0.0/1  BLOWER_AUX %
%   B3:0/15  ALARM_FLASH %
%   B3:1/1  IN_1  "Blower Aux" %
% Rung: 6 %
% When "Heater ON", setup input for Fault Catch and hold %
SOR XIC I:0.0/0 XIO B3:3/15 BST XIC I:0.0/1 NXB XIC B3:2/1 BND OTE B3:2/1 EOR
%   I:0.0/0  HEATER_ON %
%   B3:3/15  FC_RESET  "Fault Catch" %
%   I:0.0/1  BLOWER_AUX %
%   B3:2/1  FE_BLOWER_AUX  "Fault Enable" %
% Rung: 7 %
% When input is enabled, a change of state will be held untill "Heater OFF" or a "Fault Catch Reset" %
SOR XIC I:0.0/0 XIO B3:3/15 BST XIC B3:2/1 XIO I:0.0/1 NXB XIC B3:3/1 BND OTE B3:3/1 EOR
%   I:0.0/0  HEATER_ON %
%   B3:3/15  FC_RESET  "Fault Catch" %
%   B3:2/1  FE_BLOWER_AUX  "Fault Enable" %
%   I:0.0/1  BLOWER_AUX %
%   B3:3/1  FC_BLOWER_AUX  "Fault Catch" %
% Rung: 8 %
SOR XIC I:0.0/1 BST XIC I:0.0/2 NXB XIC B3:0/15 BND OTE B3:1/2 EOR
%   I:0.0/1  BLOWER_AUX %
%   I:0.0/2  EXHAUST_AUX %
%   B3:0/15  ALARM_FLASH %
%   B3:1/2  IN_2  "Exhaust Aux" %
% Rung: 9 %
% When "Heater ON", setup input for Fault Catch and hold %
SOR XIC I:0.0/0 XIO B3:3/15 BST XIC I:0.0/2 NXB XIC B3:2/2 BND OTE B3:2/2 EOR
%   I:0.0/0  HEATER_ON %
%   B3:3/15  FC_RESET  "Fault Catch" %
%   I:0.0/2  EXHAUST_AUX %
%   B3:2/2  FE_EXHAUST_AUX  "Fault Enable" %
% Rung: 10 %
% When input is enabled and the previous Fault Catch is not active, a change of state will be held untill "Heater OFF" or a "Fault Catch Reset" %
SOR XIC I:0.0/0 XIO B3:3/15 BST XIC B3:2/2 XIO I:0.0/2 NXB XIC B3:3/2 BND OTE B3:3/2 EOR
%   I:0.0/0  HEATER_ON %
%   B3:3/15  FC_RESET  "Fault Catch" %
%   B3:2/2  FE_EXHAUST_AUX  "Fault Enable" %
%   I:0.0/2  EXHAUST_AUX %
%   B3:3/2  FC_EXHAUST_AUX  "Fault Catch" %

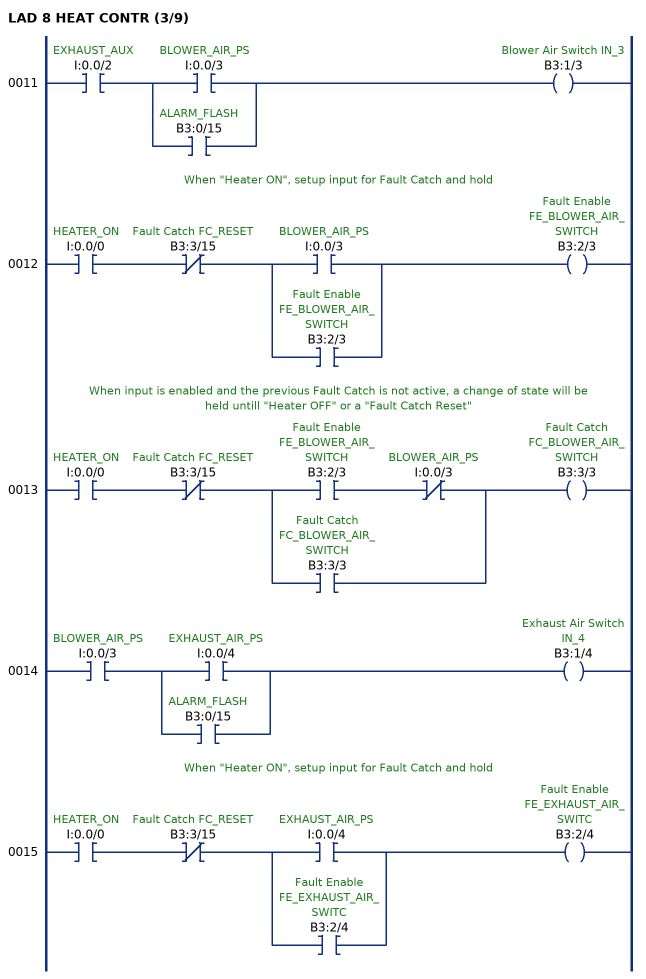
% Rung: 11 %
SOR XIC I:0.0/2 BST XIC I:0.0/3 NXB XIC B3:0/15 BND OTE B3:1/3 EOR
%   I:0.0/2  EXHAUST_AUX %
%   I:0.0/3  BLOWER_AIR_PS %
%   B3:0/15  ALARM_FLASH %
%   B3:1/3  IN_3  "Blower Air Switch" %
% Rung: 12 %
% When "Heater ON", setup input for Fault Catch and hold %
SOR XIC I:0.0/0 XIO B3:3/15 BST XIC I:0.0/3 NXB XIC B3:2/3 BND OTE B3:2/3 EOR
%   I:0.0/0  HEATER_ON %
%   B3:3/15  FC_RESET  "Fault Catch" %
%   I:0.0/3  BLOWER_AIR_PS %
%   B3:2/3  FE_BLOWER_AIR_SWITCH  "Fault Enable" %
% Rung: 13 %
% When input is enabled and the previous Fault Catch is not active, a change of state will be held untill "Heater OFF" or a "Fault Catch Reset" %
SOR XIC I:0.0/0 XIO B3:3/15 BST XIC B3:2/3 XIO I:0.0/3 NXB XIC B3:3/3 BND OTE B3:3/3 EOR
%   I:0.0/0  HEATER_ON %
%   B3:3/15  FC_RESET  "Fault Catch" %
%   B3:2/3  FE_BLOWER_AIR_SWITCH  "Fault Enable" %
%   I:0.0/3  BLOWER_AIR_PS %
%   B3:3/3  FC_BLOWER_AIR_SWITCH  "Fault Catch" %
% Rung: 14 %
SOR XIC I:0.0/3 BST XIC I:0.0/4 NXB XIC B3:0/15 BND OTE B3:1/4 EOR
%   I:0.0/3  BLOWER_AIR_PS %
%   I:0.0/4  EXHAUST_AIR_PS %
%   B3:0/15  ALARM_FLASH %
%   B3:1/4  IN_4  "Exhaust Air Switch" %
% Rung: 15 %
% When "Heater ON", setup input for Fault Catch and hold %
SOR XIC I:0.0/0 XIO B3:3/15 BST XIC I:0.0/4 NXB XIC B3:2/4 BND OTE B3:2/4 EOR
%   I:0.0/0  HEATER_ON %
%   B3:3/15  FC_RESET  "Fault Catch" %
%   I:0.0/4  EXHAUST_AIR_PS %
%   B3:2/4  FE_EXHAUST_AIR_SWITC  "Fault Enable" %

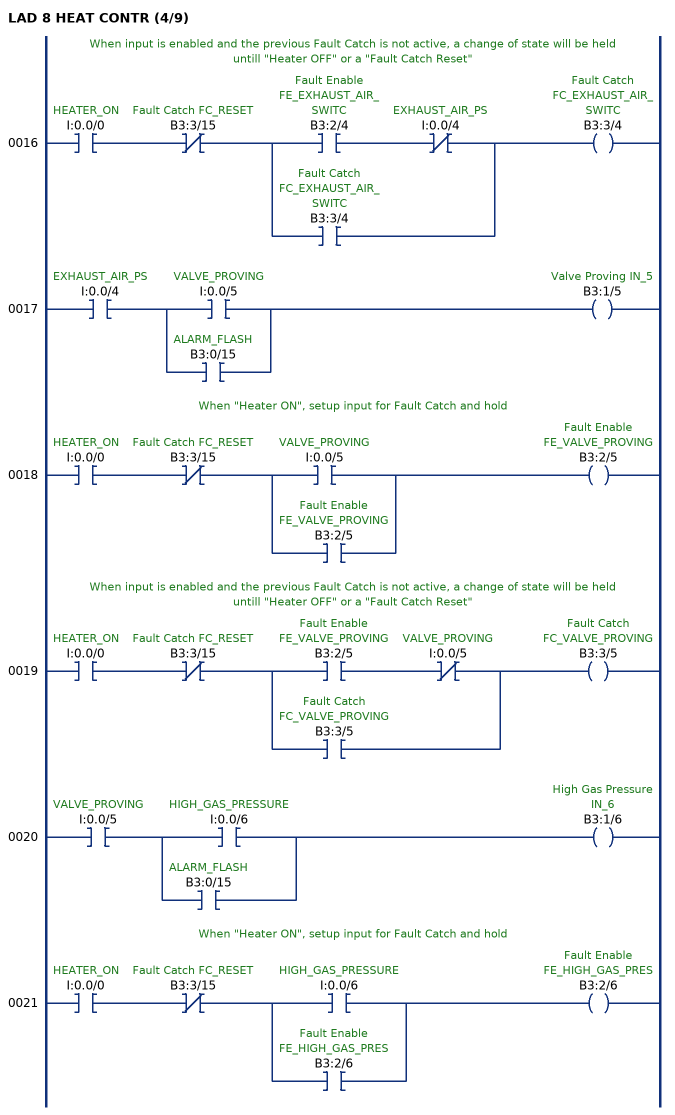
% Rung: 16 %
% When input is enabled and the previous Fault Catch is not active, a change of state will be held untill "Heater OFF" or a "Fault Catch Reset" %
SOR XIC I:0.0/0 XIO B3:3/15 BST XIC B3:2/4 XIO I:0.0/4 NXB XIC B3:3/4 BND OTE B3:3/4 EOR
%   I:0.0/0  HEATER_ON %
%   B3:3/15  FC_RESET  "Fault Catch" %
%   B3:2/4  FE_EXHAUST_AIR_SWITC  "Fault Enable" %
%   I:0.0/4  EXHAUST_AIR_PS %
%   B3:3/4  FC_EXHAUST_AIR_SWITC  "Fault Catch" %
% Rung: 17 %
SOR XIC I:0.0/4 BST XIC I:0.0/5 NXB XIC B3:0/15 BND OTE B3:1/5 EOR
%   I:0.0/4  EXHAUST_AIR_PS %
%   I:0.0/5  VALVE_PROVING %
%   B3:0/15  ALARM_FLASH %
%   B3:1/5  IN_5  "Valve Proving" %
% Rung: 18 %
% When "Heater ON", setup input for Fault Catch and hold %
SOR XIC I:0.0/0 XIO B3:3/15 BST XIC I:0.0/5 NXB XIC B3:2/5 BND OTE B3:2/5 EOR
%   I:0.0/0  HEATER_ON %
%   B3:3/15  FC_RESET  "Fault Catch" %
%   I:0.0/5  VALVE_PROVING %
%   B3:2/5  FE_VALVE_PROVING  "Fault Enable" %
% Rung: 19 %
% When input is enabled and the previous Fault Catch is not active, a change of state will be held untill "Heater OFF" or a "Fault Catch Reset" %
SOR XIC I:0.0/0 XIO B3:3/15 BST XIC B3:2/5 XIO I:0.0/5 NXB XIC B3:3/5 BND OTE B3:3/5 EOR
%   I:0.0/0  HEATER_ON %
%   B3:3/15  FC_RESET  "Fault Catch" %
%   B3:2/5  FE_VALVE_PROVING  "Fault Enable" %
%   I:0.0/5  VALVE_PROVING %
%   B3:3/5  FC_VALVE_PROVING  "Fault Catch" %
% Rung: 20 %
SOR XIC I:0.0/5 BST XIC I:0.0/6 NXB XIC B3:0/15 BND OTE B3:1/6 EOR
%   I:0.0/5  VALVE_PROVING %
%   I:0.0/6  HIGH_GAS_PRESSURE %
%   B3:0/15  ALARM_FLASH %
%   B3:1/6  IN_6  "High Gas Pressure" %
% Rung: 21 %
% When "Heater ON", setup input for Fault Catch and hold %
SOR XIC I:0.0/0 XIO B3:3/15 BST XIC I:0.0/6 NXB XIC B3:2/6 BND OTE B3:2/6 EOR
%   I:0.0/0  HEATER_ON %
%   B3:3/15  FC_RESET  "Fault Catch" %
%   I:0.0/6  HIGH_GAS_PRESSURE %
%   B3:2/6  FE_HIGH_GAS_PRES  "Fault Enable" %

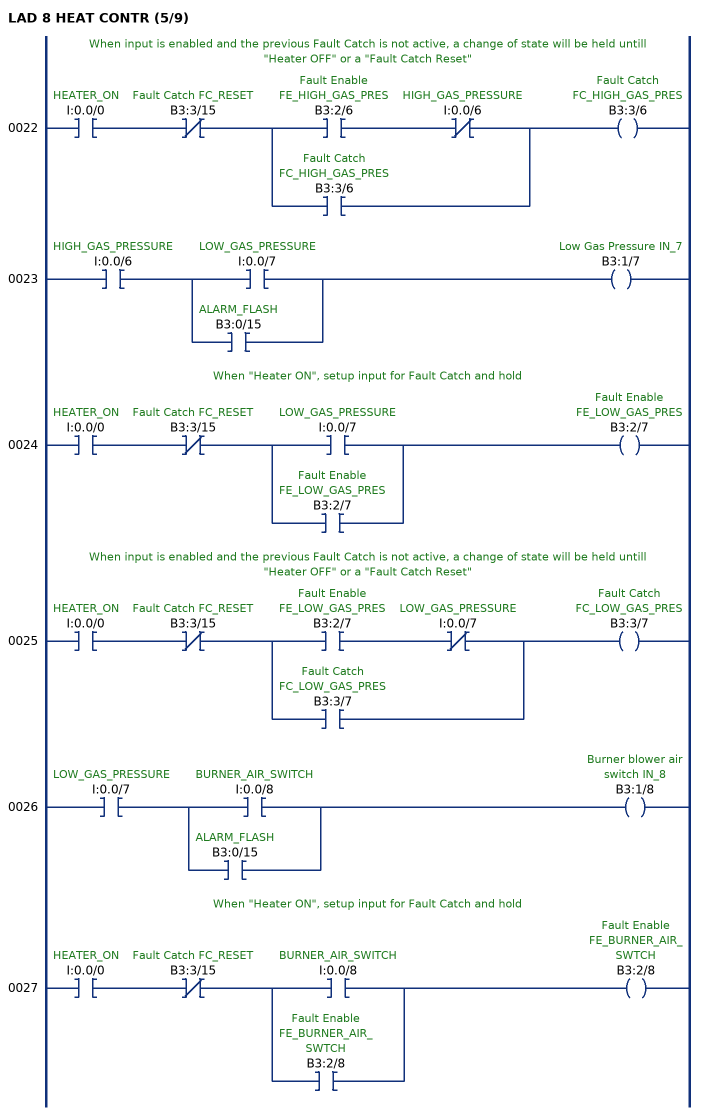
% Rung: 22 %
% When input is enabled and the previous Fault Catch is not active, a change of state will be held untill "Heater OFF" or a "Fault Catch Reset" %
SOR XIC I:0.0/0 XIO B3:3/15 BST XIC B3:2/6 XIO I:0.0/6 NXB XIC B3:3/6 BND OTE B3:3/6 EOR
%   I:0.0/0  HEATER_ON %
%   B3:3/15  FC_RESET  "Fault Catch" %
%   B3:2/6  FE_HIGH_GAS_PRES  "Fault Enable" %
%   I:0.0/6  HIGH_GAS_PRESSURE %
%   B3:3/6  FC_HIGH_GAS_PRES  "Fault Catch" %
% Rung: 23 %
SOR XIC I:0.0/6 BST XIC I:0.0/7 NXB XIC B3:0/15 BND OTE B3:1/7 EOR
%   I:0.0/6  HIGH_GAS_PRESSURE %
%   I:0.0/7  LOW_GAS_PRESSURE %
%   B3:0/15  ALARM_FLASH %
%   B3:1/7  IN_7  "Low Gas Pressure" %
% Rung: 24 %
% When "Heater ON", setup input for Fault Catch and hold %
SOR XIC I:0.0/0 XIO B3:3/15 BST XIC I:0.0/7 NXB XIC B3:2/7 BND OTE B3:2/7 EOR
%   I:0.0/0  HEATER_ON %
%   B3:3/15  FC_RESET  "Fault Catch" %
%   I:0.0/7  LOW_GAS_PRESSURE %
%   B3:2/7  FE_LOW_GAS_PRES  "Fault Enable" %
% Rung: 25 %
% When input is enabled and the previous Fault Catch is not active, a change of state will be held untill "Heater OFF" or a "Fault Catch Reset" %
SOR XIC I:0.0/0 XIO B3:3/15 BST XIC B3:2/7 XIO I:0.0/7 NXB XIC B3:3/7 BND OTE B3:3/7 EOR
%   I:0.0/0  HEATER_ON %
%   B3:3/15  FC_RESET  "Fault Catch" %
%   B3:2/7  FE_LOW_GAS_PRES  "Fault Enable" %
%   I:0.0/7  LOW_GAS_PRESSURE %
%   B3:3/7  FC_LOW_GAS_PRES  "Fault Catch" %
% Rung: 26 %
SOR XIC I:0.0/7 BST XIC I:0.0/8 NXB XIC B3:0/15 BND OTE B3:1/8 EOR
%   I:0.0/7  LOW_GAS_PRESSURE %
%   I:0.0/8  BURNER_AIR_SWITCH %
%   B3:0/15  ALARM_FLASH %
%   B3:1/8  IN_8  "Burner blower air switch" %
% Rung: 27 %
% When "Heater ON", setup input for Fault Catch and hold %
SOR XIC I:0.0/0 XIO B3:3/15 BST XIC I:0.0/8 NXB XIC B3:2/8 BND OTE B3:2/8 EOR
%   I:0.0/0  HEATER_ON %
%   B3:3/15  FC_RESET  "Fault Catch" %
%   I:0.0/8  BURNER_AIR_SWITCH %
%   B3:2/8  FE_BURNER_AIR_SWTCH  "Fault Enable" %

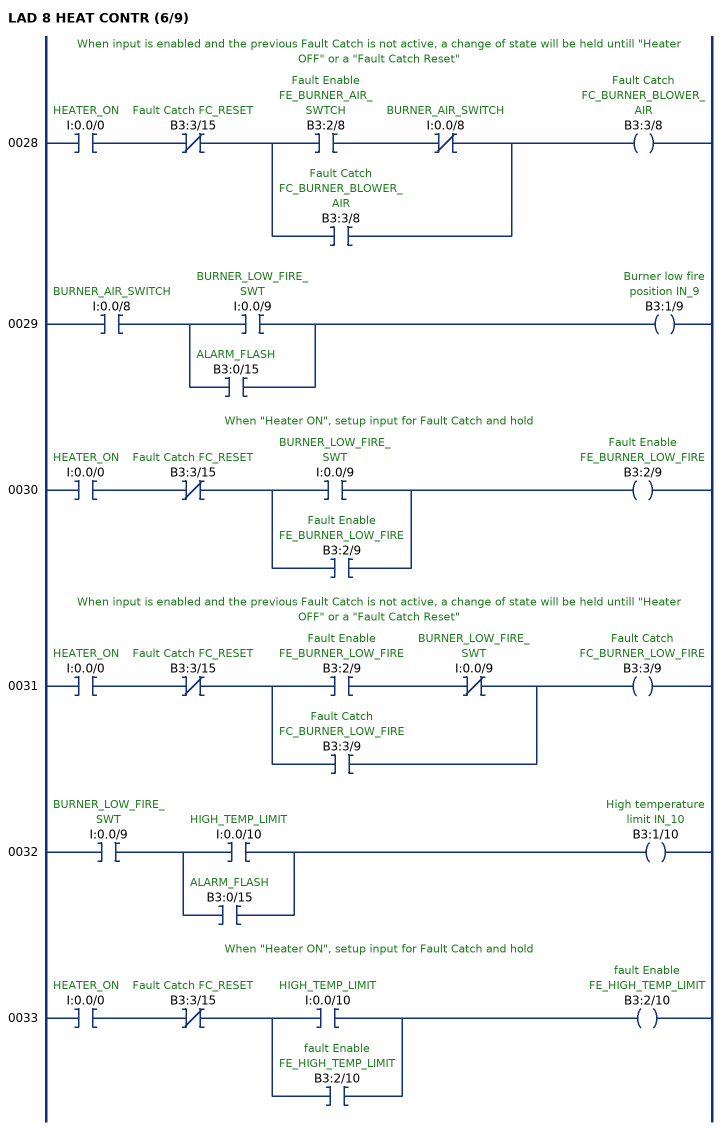
% Rung: 28 %
% When input is enabled and the previous Fault Catch is not active, a change of state will be held untill "Heater OFF" or a "Fault Catch Reset" %
SOR XIC I:0.0/0 XIO B3:3/15 BST XIC B3:2/8 XIO I:0.0/8 NXB XIC B3:3/8 BND OTE B3:3/8 EOR
%   I:0.0/0  HEATER_ON %
%   B3:3/15  FC_RESET  "Fault Catch" %
%   B3:2/8  FE_BURNER_AIR_SWTCH  "Fault Enable" %
%   I:0.0/8  BURNER_AIR_SWITCH %
%   B3:3/8  FC_BURNER_BLOWER_AIR  "Fault Catch" %
% Rung: 29 %
SOR XIC I:0.0/8 BST XIC I:0.0/9 NXB XIC B3:0/15 BND OTE B3:1/9 EOR
%   I:0.0/8  BURNER_AIR_SWITCH %
%   I:0.0/9  BURNER_LOW_FIRE_SWT %
%   B3:0/15  ALARM_FLASH %
%   B3:1/9  IN_9  "Burner low fire position" %
% Rung: 30 %
% When "Heater ON", setup input for Fault Catch and hold %
SOR XIC I:0.0/0 XIO B3:3/15 BST XIC I:0.0/9 NXB XIC B3:2/9 BND OTE B3:2/9 EOR
%   I:0.0/0  HEATER_ON %
%   B3:3/15  FC_RESET  "Fault Catch" %
%   I:0.0/9  BURNER_LOW_FIRE_SWT %
%   B3:2/9  FE_BURNER_LOW_FIRE  "Fault Enable" %
% Rung: 31 %
% When input is enabled and the previous Fault Catch is not active, a change of state will be held untill "Heater OFF" or a "Fault Catch Reset" %
SOR XIC I:0.0/0 XIO B3:3/15 BST XIC B3:2/9 XIO I:0.0/9 NXB XIC B3:3/9 BND OTE B3:3/9 EOR
%   I:0.0/0  HEATER_ON %
%   B3:3/15  FC_RESET  "Fault Catch" %
%   B3:2/9  FE_BURNER_LOW_FIRE  "Fault Enable" %
%   I:0.0/9  BURNER_LOW_FIRE_SWT %
%   B3:3/9  FC_BURNER_LOW_FIRE  "Fault Catch" %
% Rung: 32 %
SOR XIC I:0.0/9 BST XIC I:0.0/10 NXB XIC B3:0/15 BND OTE B3:1/10 EOR
%   I:0.0/9  BURNER_LOW_FIRE_SWT %
%   I:0.0/10  HIGH_TEMP_LIMIT %
%   B3:0/15  ALARM_FLASH %
%   B3:1/10  IN_10  "High temperature limit" %
% Rung: 33 %
% When "Heater ON", setup input for Fault Catch and hold %
SOR XIC I:0.0/0 XIO B3:3/15 BST XIC I:0.0/10 NXB XIC B3:2/10 BND OTE B3:2/10 EOR
%   I:0.0/0  HEATER_ON %
%   B3:3/15  FC_RESET  "Fault Catch" %
%   I:0.0/10  HIGH_TEMP_LIMIT %
%   B3:2/10  FE_HIGH_TEMP_LIMIT  "fault Enable" %

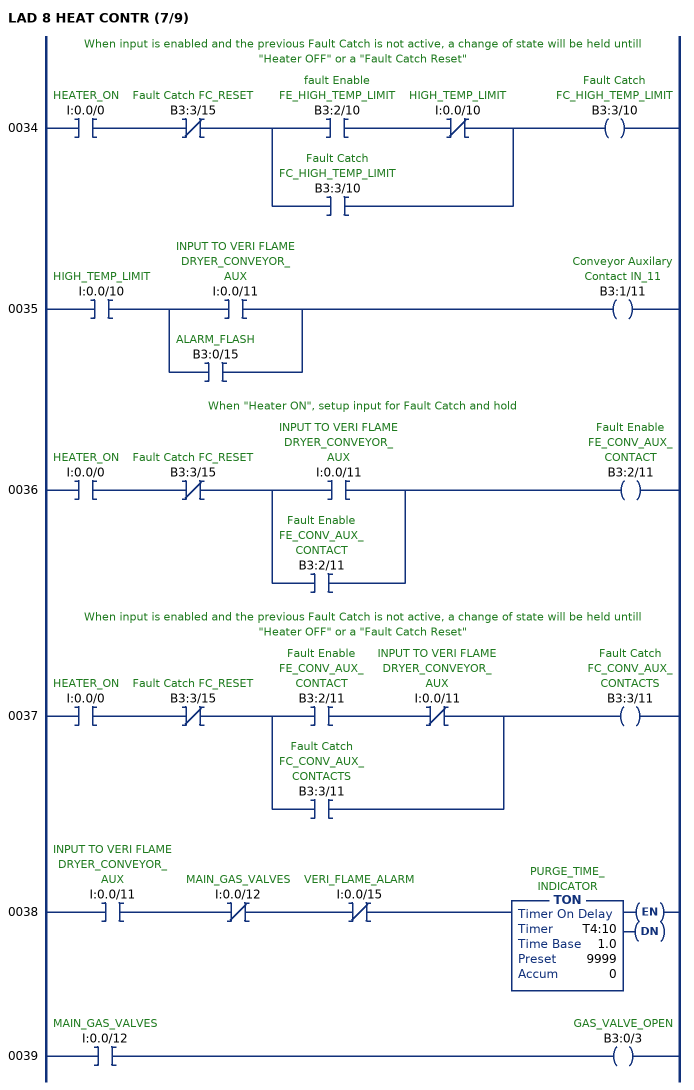
% Rung: 34 %
% When input is enabled and the previous Fault Catch is not active, a change of state will be held untill "Heater OFF" or a "Fault Catch Reset" %
SOR XIC I:0.0/0 XIO B3:3/15 BST XIC B3:2/10 XIO I:0.0/10 NXB XIC B3:3/10 BND OTE B3:3/10 EOR
%   I:0.0/0  HEATER_ON %
%   B3:3/15  FC_RESET  "Fault Catch" %
%   B3:2/10  FE_HIGH_TEMP_LIMIT  "fault Enable" %
%   I:0.0/10  HIGH_TEMP_LIMIT %
%   B3:3/10  FC_HIGH_TEMP_LIMIT  "Fault Catch" %
% Rung: 35 %
SOR XIC I:0.0/10 BST XIC I:0.0/11 NXB XIC B3:0/15 BND OTE B3:1/11 EOR
%   I:0.0/10  HIGH_TEMP_LIMIT %
%   I:0.0/11  DRYER_CONVEYOR_AUX  "INPUT TO VERI FLAME" %
%   B3:0/15  ALARM_FLASH %
%   B3:1/11  IN_11  "Conveyor Auxilary Contact" %
% Rung: 36 %
% When "Heater ON", setup input for Fault Catch and hold %
SOR XIC I:0.0/0 XIO B3:3/15 BST XIC I:0.0/11 NXB XIC B3:2/11 BND OTE B3:2/11 EOR
%   I:0.0/0  HEATER_ON %
%   B3:3/15  FC_RESET  "Fault Catch" %
%   I:0.0/11  DRYER_CONVEYOR_AUX  "INPUT TO VERI FLAME" %
%   B3:2/11  FE_CONV_AUX_CONTACT  "Fault Enable" %
% Rung: 37 %
% When input is enabled and the previous Fault Catch is not active, a change of state will be held untill "Heater OFF" or a "Fault Catch Reset" %
SOR XIC I:0.0/0 XIO B3:3/15 BST XIC B3:2/11 XIO I:0.0/11 NXB XIC B3:3/11 BND OTE B3:3/11 EOR
%   I:0.0/0  HEATER_ON %
%   B3:3/15  FC_RESET  "Fault Catch" %
%   B3:2/11  FE_CONV_AUX_CONTACT  "Fault Enable" %
%   I:0.0/11  DRYER_CONVEYOR_AUX  "INPUT TO VERI FLAME" %
%   B3:3/11  FC_CONV_AUX_CONTACTS  "Fault Catch" %
% Rung: 38 %
SOR XIC I:0.0/11 XIO I:0.0/12 XIO I:0.0/15 TON T4:10 1.0 9999 0 EOR
%   I:0.0/11  DRYER_CONVEYOR_AUX  "INPUT TO VERI FLAME" %
%   I:0.0/12  MAIN_GAS_VALVES %
%   I:0.0/15  VERI_FLAME_ALARM %
%   T4:10  PURGE_TIME_INDICATOR %
% Rung: 39 %
SOR XIC I:0.0/12 OTE B3:0/3 EOR
%   I:0.0/12  MAIN_GAS_VALVES %
%   B3:0/3  GAS_VALVE_OPEN %

